{attribute 'no_explicit_call' := 'do not call this function block directly'} 
FUNCTION_BLOCK ABSTRACT AbortableAction EXTENDS Object IMPLEMENTS IAbortableAction
VAR
	_StartRequested : BOOL;
	_AbortRequested : BOOL;
	
	_Busy : BOOL;

	_Done : BOOL;
	
	_Aborting : BOOL;	
	_Aborted : BOOL;
	_AbortReason : ERROR_MESSAGE;
	
	_Error : BOOL;	
	_ErrorMessage : ERROR_MESSAGE;	
END_VAR

{attribute 'monitoring' := 'call'}
{attribute 'OPC.UA.DA.Property' := '1'}
{attribute 'OPC.UA.DA.Access' := '1'}
PROPERTY FINAL Aborted : BOOL
GET
Aborted := _Aborted;
END_GET
END_PROPERTY

{attribute 'monitoring' := 'call'}
{attribute 'OPC.UA.DA.Property' := '1'}
{attribute 'OPC.UA.DA.Access' := '1'}
PROPERTY FINAL AbortReason : REFERENCE TO ERROR_MESSAGE
GET
AbortReason REF= _AbortReason;
END_GET
END_PROPERTY

{attribute 'monitoring' := 'call'}
{attribute 'OPC.UA.DA.Property' := '1'}
{attribute 'OPC.UA.DA.Access' := '1'}
PROPERTY FINAL Busy : BOOL
GET
Busy := _Busy OR_ELSE _Aborting;
END_GET
END_PROPERTY

{attribute 'monitoring' := 'call'}
{attribute 'OPC.UA.DA.Property' := '1'}
{attribute 'OPC.UA.DA.Access' := '1'}
PROPERTY FINAL Done : BOOL
GET
Done := _Done;
END_GET
END_PROPERTY

{attribute 'monitoring' := 'call'}
{attribute 'OPC.UA.DA.Property' := '1'}
{attribute 'OPC.UA.DA.Access' := '1'}
PROPERTY FINAL Error : BOOL
GET
Error := _Error;
END_GET
END_PROPERTY

{attribute 'monitoring' := 'call'}
{attribute 'OPC.UA.DA.Property' := '1'}
{attribute 'OPC.UA.DA.Access' := '1'}
PROPERTY FINAL ErrorMessage : REFERENCE TO ERROR_MESSAGE
GET
ErrorMessage REF= _ErrorMessage;
END_GET
END_PROPERTY

METHOD FINAL Execute 
VAR
	done : BOOL;
	
	exceptionCode : __SYSTEM.ExceptionCode;
	
	exception : IException;	
	
	errorMessage : ERROR_MESSAGE;
END_VAR
__TRY
	IF NOT Busy THEN
		IF _AbortRequested THEN
			SetAbortingState();
			
			OnAbort(TRUE, done => done);

			IF done THEN
				SetAbortedState();
			END_IF		
		ELSIF _StartRequested THEN
			SetBusyState();
			
			OnRun(TRUE, done => done);
			
			IF done THEN
				SetDoneState();
			END_IF		
		END_IF
	ELSE
		IF _Busy THEN
			OnRun(FALSE, done => done);
			
			IF done THEN
				SetDoneState();
			END_IF		
		ELSE
			OnAbort(FALSE, done => done);
			
			IF done THEN
				SetAbortedState();
			END_IF		
		END_IF
	END_IF
__CATCH(exceptionCode)
	exception := ExceptionManager.GetLastException(exceptionCode);
	
	errorMessage := exception.GetMessage();
 
	SetErrorState(errorMessage);
	
	ExceptionManager.ReThrowLastException(exceptionCode);
__ENDTRY
END_METHOD

METHOD ABSTRACT OnAbort 
VAR_INPUT
	start : BOOL;
END_VAR
VAR_OUTPUT
	done : BOOL;
END_VAR
END_METHOD

METHOD ABSTRACT OnError
END_METHOD

METHOD ABSTRACT OnRun 
VAR_INPUT
	start : BOOL;
END_VAR
VAR_OUTPUT
	done : BOOL;
END_VAR
END_METHOD

METHOD FINAL RequestAbort
VAR_INPUT 
	reason : ERROR_MESSAGE := "";
END_VAR
IF NOT Busy THEN
	RETURN;
END_IF

_AbortReason := reason;
_AbortRequested := TRUE;
END_METHOD

METHOD FINAL RequestStart
IF Busy THEN
	RETURN;
END_IF

_StartRequested := TRUE;
END_METHOD

METHOD PROTECTED FINAL SetAbortedState
_StartRequested := FALSE;
_AbortRequested := FALSE;

_Busy := FALSE;

_Done := FALSE;

_Aborting := FALSE;	
_Aborted := TRUE;

_Error := FALSE;	
_ErrorMessage := "";
END_METHOD

METHOD PROTECTED FINAL SetAbortingState
_StartRequested := FALSE;
_AbortRequested := FALSE;

_Busy := FALSE;

_Done := FALSE;

_Aborting := TRUE;	
_Aborted := FALSE;

_Error := FALSE;	
_ErrorMessage := "";
END_METHOD

METHOD PROTECTED FINAL SetBusyState
_StartRequested := FALSE;
_AbortRequested := FALSE;

_Busy := TRUE;

_Done := FALSE;

_Aborting := FALSE;	
_Aborted := FALSE;
_AbortReason := "";

_Error := FALSE;	
_ErrorMessage := "";
END_METHOD

METHOD PROTECTED FINAL SetDoneState
_StartRequested := FALSE;
_AbortRequested := FALSE;

_Busy := FALSE;

_Done := TRUE;

_Aborting := FALSE;	
_Aborted := FALSE;
_AbortReason := "";

_Error := FALSE;	
_ErrorMessage := "";
END_METHOD

METHOD PROTECTED FINAL SetErrorState
VAR_IN_OUT CONSTANT
	errorMessage : ERROR_MESSAGE;
END_VAR
_StartRequested := FALSE;
_AbortRequested := FALSE;

_Busy := FALSE;

_Done := FALSE;

_Aborting := FALSE;	
_Aborted := FALSE;
_AbortReason := "";

_Error := TRUE;	
_ErrorMessage := errorMessage;
END_METHOD

END_FUNCTION_BLOCK

(* stored: Version 1.1.0.1
   POU AbortableAction: Id {3fcb82bf-fcc2-4c60-ab58-32776172ce5b}, SpecialFunc None
   Folder Members to override: Id {76112447-5878-4246-92fb-0910ffa3ef2d}
   Folder Service members: Id {6b1a5589-8d7c-4542-877b-5fcd2d9b2fbd}
   Property Aborted: Id {205fba08-26d2-4312-a96e-e17dee6c923f}
   Get Get: Id {9f8851fa-4d24-41c2-b7cf-fd9ecc9bdb84}
   Property AbortReason: Id {62b5d978-3b39-4864-a514-bb07423cf0e2}
   Get Get: Id {e89b4f7e-5119-407b-92c1-18a61068d8bb}
   Property Busy: Id {dda6cb05-0e58-4715-8fa9-9ed4428ca958}
   Get Get: Id {ac4bced3-fa18-48d8-a5d4-4beba0226ec1}
   Property Done: Id {b95d743b-c72e-4bcb-a404-c7e3e4a6a37e}
   Get Get: Id {bfaa887d-c314-4518-a171-41d0308d56ff}
   Property Error: Id {3d54590f-9d24-46b4-9724-32260ce4207a}
   Get Get: Id {998b8321-1744-4a0a-b9cf-78a20c7dc6e5}
   Property ErrorMessage: Id {e92b95ec-4a2f-46a9-85eb-1f48df75a257}
   Get Get: Id {82e42fe0-1017-4cc0-a630-23020b73322e}
   Method Execute: Id {356dfaf1-5836-4634-88c3-9adf266fe2b8}
   Method OnAbort: Id {bd8eb179-c550-42d5-a679-2b68c1503c0e}
   Method OnError: Id {c12cd4b4-6b5e-40a4-9547-4538d1fad656}
   Method OnRun: Id {a15599f5-e9ad-4bc1-b827-e975fc966d86}
   Method RequestAbort: Id {f4d5eddb-0774-4410-8518-af02c1510410}
   Method RequestStart: Id {5e4f958e-3441-449c-a3ee-2bfa2bc2b0b1}
   Method SetAbortedState: Id {fac00809-31d6-4f90-8e02-b442214ce266}
   Method SetAbortingState: Id {dc660dfe-c65d-4d91-bb97-ccc531a7b715}
   Method SetBusyState: Id {8ba032d1-b467-4f29-94d8-e5d440995321}
   Method SetDoneState: Id {5a91bd28-905f-4ff0-ac15-4afd240589a6}
   Method SetErrorState: Id {1017a81e-af2a-4781-bfcb-fe042f84da43} *)
